FUNCTION_BLOCK FB_SetTimeModel
VAR_INPUT
END_VAR
VAR_OUTPUT
END_VAR
VAR
	nCallCount : UINT;
	stTimeModel : ST_TimeModelDataType;
END_VAR

{attribute 'TcRpcEnable' := '1'}
METHOD Abort : HRESULT
VAR_INPUT
END_VAR
END_METHOD

PROPERTY bBusy : BOOL
GET
END_GET
SET
END_SET
END_PROPERTY

{attribute 'TcRpcEnable' := '1'}
METHOD CheckState : HRESULT
VAR_INPUT
	hdl : UDINT;
END_VAR
END_METHOD

PROPERTY hrError : HRESULT
GET
END_GET
SET
END_SET
END_PROPERTY

{attribute 'TcRpcEnable' := '1'}
METHOD Start : HRESULT
VAR_INPUT
	TimeModel : ST_TimeModelDataType;
END_VAR
nCallCount := nCallCount + 1;
stTimeModel := TimeModel;
END_METHOD

END_FUNCTION_BLOCK

(* stored: Version 1.1.0.1, ProductVersion 3.1.4024.3
   POU FB_SetTimeModel: Id {bad34322-1359-4aed-9351-5dfc9a9e6716}, SpecialFunc None
   Method Abort: Id {92559d52-4085-4e05-a28a-7b73631ab0ca}
   Property bBusy: Id {63d8a30a-b061-4fd8-82f6-557644412f1e}
   Get Get: Id {3970d8d3-bba0-4710-b6c0-b1cf34a25391}
   Set Set: Id {2288a6de-daac-4f5c-b566-b3b3c85d9abe}
   Method CheckState: Id {c6d51e06-c163-4759-9e3a-190ae768e9bb}
   Property hrError: Id {b43360b5-942a-426e-b4d4-2c1d61dda952}
   Get Get: Id {cc03406c-4ba8-4b3c-8afb-472a8bf4c7ec}
   Set Set: Id {d7f5047a-e36d-450e-97cb-64fd4229f14d}
   Method Start: Id {f70119c4-38cb-4f91-80e0-334b28876d0d} *)
